// TIA Portal V19 export
DATA_BLOCK "Actions"   // DB3
{ S7_Optimized_Access := 'TRUE' }
// stored: MemoryReserve 100
   VAR
      Action_AirComprID1 : String := 'Check that no emergency stop has been depressed. If it has, check why. The machine is now ready to start with the Unit On button. The alarm is reset automatically when the cause is removed (logically controlled).';
      TextList : DWord;
      Trigger : UInt;
      Ack : Bool;
   END_VAR
BEGIN
END_DATA_BLOCK
